TYPE ST_ModuleConfigurationStatus :
STRUCT
	Ready : BOOL;
	Error : BOOL;
	ErrorCode : E_ConfigValueError;
	ErrorMessage : STRING(255);
	ErrorSource : STRING(255);
END_STRUCT
END_TYPE

(* stored: Version 1.1.0.1, ProductVersion 3.1.4026.18
   DUT ST_ModuleConfigurationStatus: Id {d2929b2a-eba4-4856-92c9-648229124038} *)
